TYPE ST_STATION_GEAR_PARAMETER :
STRUCT
  eDistance           : E_STATION_GEAR_DISTANCE_AXIS; // follow which leader?
  rSyncDistance       : LREAL := 100.0;               // synchrone distance while the mover is geared in
  rMinDistanceToSync  : LREAL := 100.0;               // minimum distance for mover to get nSync with the Master
END_STRUCT
END_TYPE

(* stored: Version 1.1.0.1, ProductVersion 3.1.4026.18
   DUT ST_STATION_GEAR_PARAMETER: Id {67b2479a-fca5-4563-853a-a1e80ec89546} *)
